(* PLC project v0.6.04_CycleSemiAuto.project, CODESYS CODESYS V3.5 SP19 Patch 1 *)
(* stored: creationDateTime 2026-08-11T14:02:33.665714, modificationDateTime 2026-08-11T14:02:33.665714 *)

(* ═══════════════════════════════════════════════════════════════ 🎮 ST_BucketCmd — Commandes IHM pour la benne (M2) ═══════════════════════════════════════════════════════════════ *)
TYPE ST_BucketCmd : STRUCT
  BtnOpen : BOOL;  (* 🪣 Bouton commande ouverture *)
  BtnClose : BOOL;  (* 🪣 Bouton commande fermeture *)
  BtnReset : BOOL;  (* 🔑 Acquittement défaut benne *)
  BtnConfirmOpenPos : BOOL;  (* 🆕 Référencement benne position ouverte (mise en service) — confirmation pure, aucun mouvement *)
  BtnConfirmClosePos : BOOL;  (* 🆕 Référencement benne position fermée (mise en service) — confirmation pure, aucun mouvement *)
  TglManualBucketLimits : BOOL := TRUE;  (* 🆕 2026-08-07 (18) : mode pilotage unitaire M2 "sécurisé" (demande client) -- actif uniquement en SelJoystickWinch=2 (unitaire M2). Si TRUE : borne le déplacement entre les positions ouvert/fermé configurées (OffsetOpenM/OffsetCloseM relatif à M1, mêmes bornes que FB_Bucket) ET plafonne la vitesse au palier 1, sans passer par instBucket (pas de mémorisation CloseReq/OpenReq, jogging libre borné). Défaut FALSE : pilotage unitaire M2 sans limite dédiée. 🆕 2026-08-07 (18bis) : défaut TRUE (demande client) -- pilotage unitaire M2 borné + palier 1 par défaut *)
END_STRUCT;
END_TYPE
